FUNCTION_BLOCK L3_MMCore (* Machine manager core *)
  (* Standard: 61499-2; Description: This FB handles the machine state vectors. It determines, periodically, which PP can take each machine in the system. *)
  (* Version 0.0, 2014-10-06, EQUEROL, UJI *)
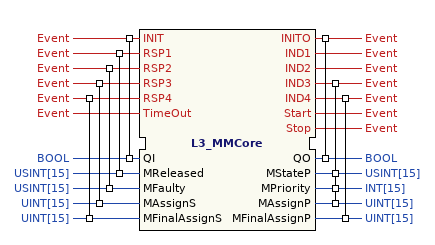
  EVENT_INPUT
    INIT WITH QI; (* Initialization Request *)
    RSP1 WITH MReleased; (* IND1 Response *)
    RSP2 WITH MFaulty; (* IND2 response *)
    RSP3 WITH MAssignS; (* IND3 response *)
    RSP4 WITH MFinalAssignS; (* IND4 response *)
    TimeOut; (* cyclic execution timeout *)
  END_EVENT
  EVENT_OUTPUT
    INITO WITH QO; (* Initialization Confirm *)
    IND1; (* Requests released machines vector *)
    IND2; (* Requests faulty machines vector *)
    IND3 WITH MStateP, MPriority, MAssignP; (* Request a check of the needed machines *)
    IND4 WITH MFinalAssignP; (* Requests the star of the machines allocation *)
    Start; (* Start timeout counter *)
    Stop; (* Stop timeout counter *)
  END_EVENT
  VAR_INPUT
    QI : BOOL; (* Input event qualifier *)
    MReleased : ARRAY [0..14] OF USINT; (* Released machines vector *)
    MFaulty : ARRAY [0..14] OF USINT; (* Faulty machines vector *)
    MAssignS : ARRAY [0..14] OF UINT; (* Machine-PP assignation vector *)
    MFinalAssignS : ARRAY [0..14] OF UINT; (* Machine-PP assignation vector *)
  END_VAR
  VAR_OUTPUT
    QO : BOOL; (* Output event qualifier *)
    MStateP : ARRAY [0..14] OF USINT; (* Machine State vector *)
    MPriority : ARRAY [0..14] OF INT; (* Machine allocations priority vector *)
    MAssignP : ARRAY [0..14] OF UINT; (* Machine-PP assignation vector *)
    MFinalAssignP : ARRAY [0..14] OF UINT; (* Machine-PP assignation vector *)
  END_VAR
  VAR
    MState : ARRAY [0..14] OF USINT := [0,0,0,0,0,0,0,0,0,0,0,0,0,0,0]; (* Internal vector to hold machine state *)
    i : USINT; (* Loop variable *)
    MachineCounter : USINT := 0; (* Internal Variable *)
  END_VAR
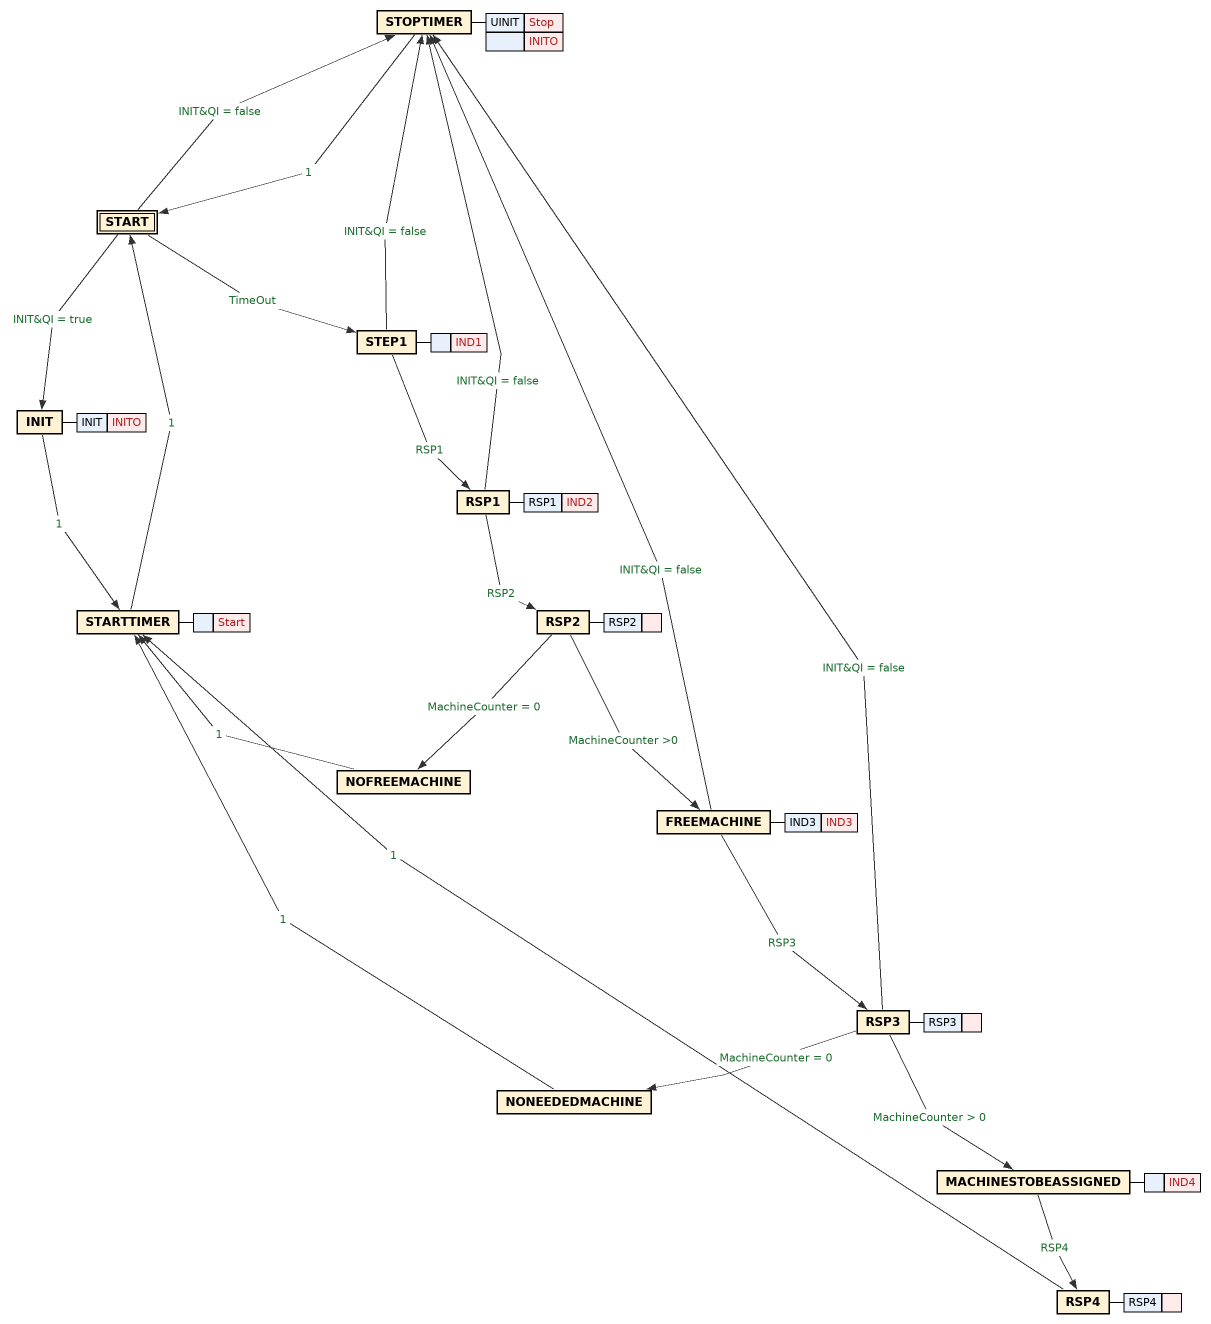
  EC_STATES
    START; (* Initial State *)
    INIT : INIT -> INITO; (* Initialization *)
    STEP1 : -> IND1; (* Normal execution *)
    RSP1 : RSP1 -> IND2;
    NOFREEMACHINE;
    RSP2 : RSP2;
    FREEMACHINE : IND3 -> IND3;
    RSP3 : RSP3;
    RSP4 : RSP4;
    STARTTIMER : -> Start;
    STOPTIMER : UINIT -> Stop, -> INITO;
    MACHINESTOBEASSIGNED : -> IND4;
    NONEEDEDMACHINE;
  END_STATES
  EC_TRANSITIONS
    STEP1 TO RSP1 := RSP1;
    RSP2 TO FREEMACHINE := MachineCounter >0;
    RSP2 TO NOFREEMACHINE := MachineCounter = 0;
    FREEMACHINE TO RSP3 := RSP3;
    RSP1 TO RSP2 := RSP2;
    START TO STEP1 := TimeOut;
    STARTTIMER TO START := 1;
    NOFREEMACHINE TO STARTTIMER := 1;
    START TO STOPTIMER := INIT&QI = false;
    STOPTIMER TO START := 1;
    STEP1 TO STOPTIMER := INIT&QI = false;
    RSP1 TO STOPTIMER := INIT&QI = false;
    FREEMACHINE TO STOPTIMER := INIT&QI = false;
    RSP3 TO STOPTIMER := INIT&QI = false;
    RSP4 TO STARTTIMER := 1;
    RSP3 TO NONEEDEDMACHINE := MachineCounter = 0;
    RSP3 TO MACHINESTOBEASSIGNED := MachineCounter > 0;
    MACHINESTOBEASSIGNED TO RSP4 := RSP4;
    NONEEDEDMACHINE TO STARTTIMER := 1;
    START TO INIT := INIT&QI = true;
    INIT TO STARTTIMER := 1;
  END_TRANSITIONS
  ALGORITHM INIT IN ST: (* Initialization algorithm *)
(*Reset internal variables*)
FOR i := 0 TO 14 DO
	MState[i] := 0;
	MAssignP[i] := 0;
	MPriority[i] := 0;
END_FOR;
MachineCounter := 0;
QO := TRUE;
  END_ALGORITHM
  ALGORITHM RSP1 IN ST: (* Algorithm to update released machines *)
(*This algo is in charge of updating the released machines since last time that CORE sequence was executed*)
FOR i := 0 TO 14 DO
	IF MReleased[i] = 2 THEN
		(*Machine was released*)
		MState[i] := 2;
	END_IF;
END_FOR;
  END_ALGORITHM
  ALGORITHM RSP2 IN ST: (* Algorithm to update breakdown machines *)
MachineCounter := 0;
FOR i := 0 TO 14 DO
	IF MFaulty[i] = 1 THEN
		(*Machine breakdown*)
		MState[i] := 1;
	ELSIF MFaulty[i] = 2 THEN
		(*Machine was repaired*)
		MState[i] := 2;
	END_IF;

	IF MState[i]  = 2 THEN
		MachineCounter := MachineCounter +1;
	END_IF;
END_FOR;
  END_ALGORITHM
  ALGORITHM RSP3 IN ST: (* Algorithm in charge of verifying if any PP needs to use any of the unused machines *)
(*MAssignS[i] contains 0 if the machine wasn't requested, otherwise the ID of the PP that requested the machine*)
MachineCounter := 0;
FOR i := 0 TO 14 DO
	MFinalAssignP[i] := MAssignS[i];
	IF MFinalAssignP[i] <> 0 THEN
		MState[i] := 3;
		MachineCounter := MachineCounter +1;
	END_IF;
END_FOR;
  END_ALGORITHM
  ALGORITHM RSP4 IN ST: (* Updates MSate if any machine was correctly assigned *)
(*MFinalAssignS[i] is 0 if the machine assignation succeed, otherwise the assignation failed*)
FOR i := 0 TO 14 DO
	IF MFinalAssignS[i] = 0 THEN
		(*Assignation succeed*)
		MState[i] := 4;
	ELSE
		(*Assignation failed, mark machine as free, will handle its real state in next cycle*)
		MState[i] := 2;
	END_IF;
END_FOR;
  END_ALGORITHM
  ALGORITHM UINIT IN ST: (* Uninitalisation algo *)
QO := FALSE;
  END_ALGORITHM
  ALGORITHM IND3 IN ST: (* Algo to reset vectors before starting the negotiation process *)
FOR i := 0 TO 14 DO
	MStateP[i] := MState[i] ;
	MAssignP[i] := 0;
	MPriority[i] := 32766;
END_FOR;
  END_ALGORITHM
END_FUNCTION_BLOCK
